FUNCTION_BLOCK FB_Example
VAR
    bStart : BOOL;
    iSpeed : INT;
END_VAR
BEGIN
MyMotor(
    Start := bStart,
    Speed := iSpeed
);
END_FUNCTION_BLOCK
